PROGRAM Alarm_Flag
VAR
END_VAR

// NETWORK 1

END_PROGRAM

(* stored: Version 1.1.0.1, ProductVersion 3.1.4024.0
   POU Alarm_Flag: Id {adacf555-eefc-4dec-baf0-d66f9d68e5aa}, SpecialFunc None *)
